FUNCTION_BLOCK FB_TestSuiteGroup
VAR
    fbTestSuite3Instance1 : FB_TestSuite3;
END_VAR

END_FUNCTION_BLOCK

(* stored: Version 1.1.0.1, ProductVersion 3.1.4024.12
   POU FB_TestSuiteGroup: Id {0f5f66b5-a14b-4e9c-b940-1dbbd259c922}, SpecialFunc None *)
